// SIMATIC STEP 7 (V5.x) project N2021Andres
// CPU: CPU 314C-2 DP
// station: Hardware
// station: SIMATIC 300 maestro
// station: P_ADR_BUS
// station: P_ADR_BUS
// station: Configuración
// program: Programa S7(1)

SYMBOL_TABLE
"Con_flujo"	C 12	COUNTER
"TempAguaFria"	C 13	COUNTER
"TempAguaCAliente"	C 14	COUNTER
"TempVapor"	C 15	COUNTER
"TempCondensados"	C 16	COUNTER
"EntradasING"	DB 1	DB 1
"Datos1Hp"	DB 3	DB 3	// Datos leidos y enviados al variador de 1 Hp
"Datos2HP"	DB 4	DB 4	// Datos leidos y enviados al variador de 2 Hp
"DatosVarpH"	DB 6	DB 6	// Datos leidos y enviados al variador de 1 Hp
"DatosVarReactor"	DB 7	DB 7	// Datos leidos y enviados al variador de 1 Hp
"CONT_C"	FB 41	FB 41	// Continuous Control
"Escalizaciones"	FC 1	FC 1
"Alarmas"	FC 2	FC 2
"var1hp"	FC 3	FC 3
"var2hp"	FC 4	FC 4
"VarReactor"	FC 5	FC 5
"VarpH"	FC 6	FC 6
"DP_SEND"	FC 15	FC 15	// DP-SEND-Function for  SIMATIC NET CPs
"FT_In"	I 0.0	BOOL
"nivelAltoAlim"	I 2.0	BOOL
"nivelbajoAlim"	I 2.1	BOOL
"termico1hp"	I 2.3	BOOL
"termico2hp"	I 2.4	BOOL
"H_Emergencia"	I 2.5	BOOL
"start1hp"	M 1.0	BOOL
"stop1hp"	M 1.1	BOOL
"recFall1hp"	M 1.2	BOOL
"start2hp"	M 1.3	BOOL
"stop2hp"	M 1.4	BOOL
"recFalla2hp"	M 1.5	BOOL
"ResetSPNivel"	M 1.6	BOOL
"siempreOff"	M 2.0	BOOL
"siempreon"	M 2.1	BOOL
"Cascada"	M 2.2	BOOL
"manpid1"	M 2.3	BOOL
"manpid2"	M 2.4	BOOL
"manpid3"	M 2.5	BOOL
"M_ALLTKpeq"	M 3.0	BOOL
"M_AHLTKpeq"	M 3.1	BOOL
"M_Termico1HP"	M 3.2	BOOL
"M_LT_alto"	M 3.3	BOOL
"M_Termico2HP"	M 3.4	BOOL
"M_H.Emerg"	M 3.5	BOOL
"M_AlarmaSobrepresiòn"	M 3.6	BOOL
"AlamaBitporpresion"	M 3.7	BOOL
"resetTotalFlujo"	M 5.0	BOOL
"startReactor"	M 184.0	BOOL
"StopReactor"	M 184.1	BOOL
"RecFallaReactor"	M 184.2	BOOL
"StartpH"	M 184.3	BOOL
"StoppH"	M 184.4	BOOL
"RecFallapH"	M 184.5	BOOL
"FT_Aire_mA"	MD 132	REAL	// señal escalizada en mA del FT de aire a la salida del tanque
"FlujoAireOutLPM"	MD 136	REAL	// flujo de aire medido con el sensor portatil a la salida de la valvula prop
"VoltReactor"	MD 140	REAL
"CorrReactor"	MD 144	REAL
"FreReactor"	MD 148	REAL
"VoltpH"	MD 152	REAL
"CorrpH"	MD 156	REAL
"FrepH"	MD 160	REAL
"Tiempo"	MD 164	REAL
"Total_litros"	MD 172	REAL
"ohmiosPT100"	MD 176	REAL	// ohmios equivalntes para la temperatura db1.dbd40
"flujo_In_lpm"	MD 180	REAL
"Flujo_Out_lpm"	MD 184	REAL
"fre2hp"	MD 188	REAL
"vol2hp"	MD 192	REAL
"corr2hp"	MD 196	DWORD
"fre1hp"	MD 200	DWORD
"vol1hp"	MD 204	REAL
"corr1hp"	MD 208	DWORD
"LTmA"	MD 212	REAL
"FTmA"	MD 216	REAL
"mA_A_IP"	MD 220	REAL
"mA_A_Valve_Prop"	MD 224	REAL
"FrecuenciaDint2"	MD 228	DINT
"pTmA"	MD 232	REAL
"PT_Out_mA"	MD 236	REAL
"LTpsig"	MD 240	REAL
"PulsosTotal"	MD 244	REAL
"PulsosRata"	MD 248	REAL
"FrecuenciaDint"	MD 252	DINT
"FrecuenciaReal"	MD 256	REAL
"erroresfc"	MW 64	WORD
"fre2hpref"	MW 98	WORD
"fre1hpref"	MW 100	WORD
"freReactorref"	MW 102	WORD
"frepHref"	MW 104	WORD
"CYC_INT2"	OB 32	OB 32	// Cyclic Interrupt 2
"CYC_INT3"	OB 33	OB 33	// Cyclic Interrupt 3
"CYC_INT6"	OB 36	OB 36	// Cyclic Interrupt 6
"CYC_INT8"	OB 38	OB 38	// Cyclic Interrupt 8
"LTint"	PIW 50	INT	// FT ultrasonido de nivel rango 0-60cms
"PTint"	PIW 52	INT	// PT en el tanque rango  0-600mBar
"FTint"	PIW 54	INT	// FT en tuberia rango 0-60LPM
"FT_Aire"	PIW 56	INT	// FT flujo aire portatil 0-20 SLPM
"libre1"	PIW 58	WORD
"IP"	PQW 50	WORD
"PropValve"	PQW 52	WORD
"BalisaLuminosa"	Q 0.3	BOOL
"FREQUENC"	SFB 48	SFB 48	// Frequency measurement module
"WR_REC"	SFC 58	SFC 58	// Write Data Record
"com"	VAT 1	
END_SYMBOL_TABLE

// FB 41: know-how protected block, not included

FUNCTION "Escalizaciones" : VOID	// FC 1
VERSION : 0.1
VAR_TEMP
  TEMP0 : DINT ;
  TEMP1 : REAL ;
  temp2 : DINT ;
END_VAR
BEGIN
NETWORK
TITLE = Escalizamos el transmisor de nivel en cms y en mA
      A     "siempreOff";
      =     L 12.0;
      BLD   103;
      A(;
      A     "siempreOff";
      =     L 12.1;
      BLD   103;
      CALL  FC 105 (
           $1                       := P#P 50.0,
           $2                       := L#1114898432,
           $3                       := L#0,
           $4                       := L 12.1,
           $5                       := "erroresfc",
           $6                       := DB10.DBD 10);
      A     BR;
      );
      JNB   _001;
      CALL  FC 105 (
           $1                       := P#P 50.0,
           $2                       := L#1101004800,
           $3                       := L#1082130432,
           $4                       := L 12.0,
           $5                       := "erroresfc",
           $6                       := "LTmA");
_001: NOP   0;
NETWORK
TITLE = Escalizamos el transmisor de presiòn en mbar, en psig y en mA
      A     "siempreOff";
      =     L 12.0;
      BLD   103;
      A(;
      A     "siempreOff";
      =     L 12.1;
      BLD   103;
      CALL  FC 105 (
           $1                       := P#P 52.0,
           $2                       := L#1142292480,
           $3                       := L#0,
           $4                       := L 12.1,
           $5                       := "erroresfc",
           $6                       := DB9.DBD 10);
      A     BR;
      );
      JNB   _002;
      CALL  FC 105 (
           $1                       := P#P 52.0,
           $2                       := L#1101004800,
           $3                       := L#1082130432,
           $4                       := L 12.0,
           $5                       := "erroresfc",
           $6                       := "pTmA");
_002: NOP   0;
NETWORK
TITLE = Escalizamos el transmisor de flujo ultrasonido en lpm y mA
      A     "siempreOff";
      =     L 12.0;
      BLD   103;
      A(;
      A     "siempreOff";
      =     L 12.1;
      BLD   103;
      CALL  FC 105 (
           $1                       := P#P 54.0,
           $2                       := L#1101004800,
           $3                       := L#1082130432,
           $4                       := L 12.1,
           $5                       := "erroresfc",
           $6                       := "FTmA");
      A     BR;
      );
      JNB   _003;
      CALL  FC 105 (
           $1                       := P#P 54.0,
           $2                       := L#1114636288,
           $3                       := L#0,
           $4                       := L 12.0,
           $5                       := "erroresfc",
           $6                       := DB11.DBD 10);
_003: NOP   0;
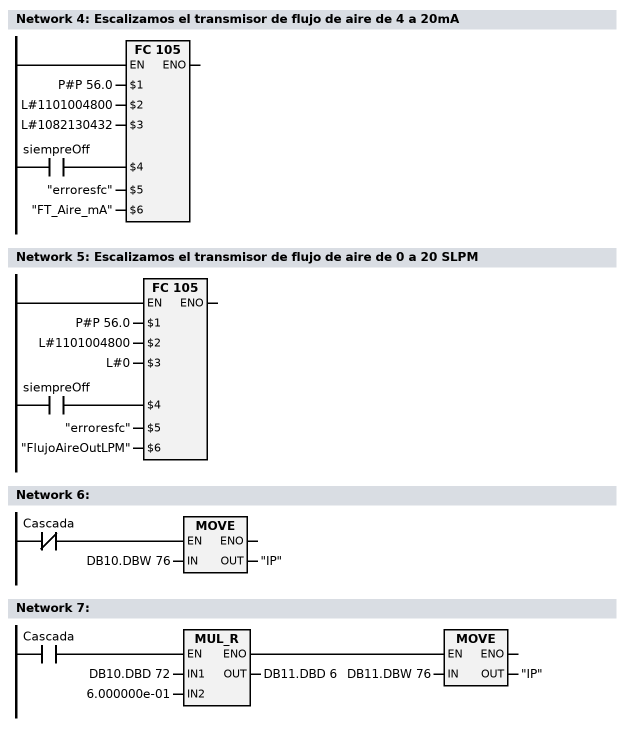
NETWORK
TITLE = Escalizamos el transmisor de flujo de aire de 4 a 20mA
      A     "siempreOff";
      =     L 12.0;
      BLD   103;
      CALL  FC 105 (
           $1                       := P#P 56.0,
           $2                       := L#1101004800,
           $3                       := L#1082130432,
           $4                       := L 12.0,
           $5                       := "erroresfc",
           $6                       := "FT_Aire_mA");
      NOP   0;
NETWORK
TITLE = Escalizamos el transmisor de flujo de aire de 0 a 20 SLPM
      A     "siempreOff";
      =     L 12.0;
      BLD   103;
      CALL  FC 105 (
           $1                       := P#P 56.0,
           $2                       := L#1101004800,
           $3                       := L#0,
           $4                       := L 12.0,
           $5                       := "erroresfc",
           $6                       := "FlujoAireOutLPM");
      NOP   0;
NETWORK
TITLE =
//Si es control de nivel llevamos la salida al IP1
      AN    "Cascada";
      JNB   _004;
      L     DB10.DBW 76;
      T     "IP";
_004: NOP   0;
NETWORK
TITLE =
//LLevamos la salida del control de nivel como setPoint al control de flujo y la 
//salida del control de flujo a la salida fisica
//
      A(;
      A     "Cascada";
      JNB   _005;
      L     DB10.DBD 72;
      L     6.000000e-01;
      *R;
      T     DB11.DBD 6;
      AN    OV;
      SAVE;
      CLR;
_005: A     BR;
      );
      JNB   _006;
      L     DB11.DBW 76;
      T     "IP";
_006: NOP   0;
END_FUNCTION

FUNCTION "Alarmas" : VOID	// FC 2
VERSION : 0.1
BEGIN
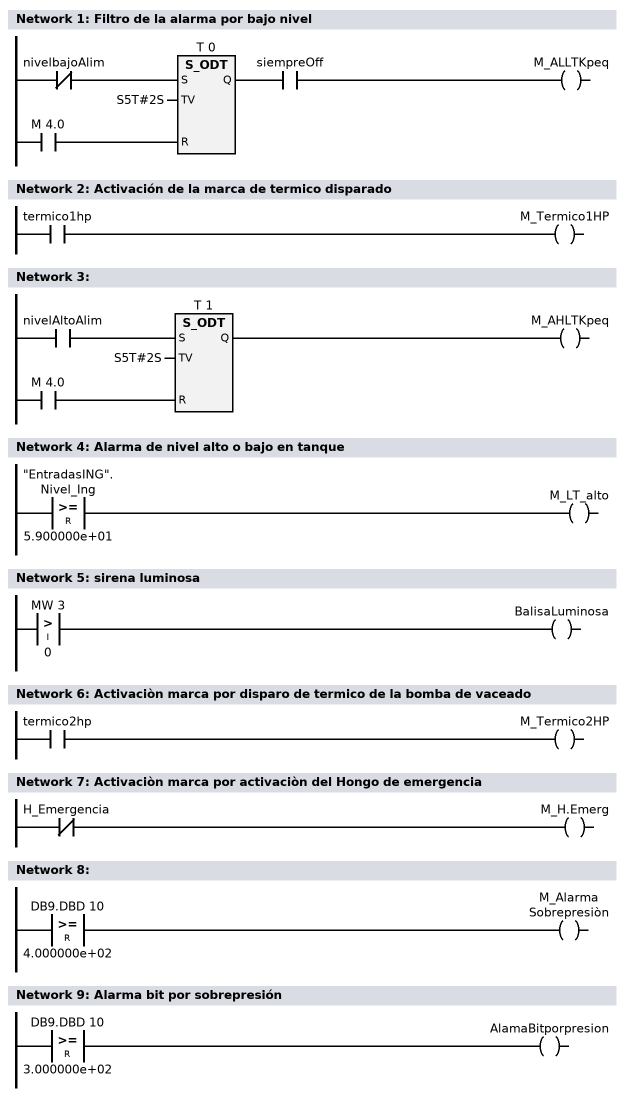
NETWORK
TITLE = Filtro de la alarma por bajo nivel
      A(;
      AN    "nivelbajoAlim";
      L     S5T#2S;
      SD    T 0;
      A     M 4.0;
      R     T 0;
      NOP   0;
      NOP   0;
      A     T 0;
      );
      A     "siempreOff";
      =     "M_ALLTKpeq";
NETWORK
TITLE = Activación de la marca de termico disparado
      A     "termico1hp";
      =     "M_Termico1HP";
NETWORK
TITLE =
//Filtro de la alarma por alto nivel
      A     "nivelAltoAlim";
      L     S5T#2S;
      SD    T 1;
      A     M 4.0;
      R     T 1;
      NOP   0;
      NOP   0;
      A     T 1;
      =     "M_AHLTKpeq";
NETWORK
TITLE = Alarma de nivel alto o bajo en tanque
      L     "EntradasING".Nivel_Ing;
      L     5.900000e+01;
      >=R;
      =     "M_LT_alto";
NETWORK
TITLE = sirena luminosa
      L     MW 3;
      L     0;
      >I;
      =     "BalisaLuminosa";
NETWORK
TITLE = Activaciòn marca por disparo de termico de la bomba de vaceado
      A     "termico2hp";
      =     "M_Termico2HP";
NETWORK
TITLE = Activaciòn marca por activaciòn del Hongo de emergencia
      AN    "H_Emergencia";
      =     "M_H.Emerg";
NETWORK
TITLE =
      L     DB9.DBD 10;
      L     4.000000e+02;
      >=R;
      =     "M_AlarmaSobrepresiòn";
NETWORK
TITLE = Alarma bit por sobrepresión
      L     DB9.DBD 10;
      L     3.000000e+02;
      >=R;
      =     "AlamaBitporpresion";
END_FUNCTION

FUNCTION "var1hp" : VOID	// FC 3
TITLE = Lectura y escritura de datos en el variador de 1Hp
VERSION : 0.1
VAR_TEMP
  temp1_1 : INT ;
  freRef : INT ;
  temp1 : DINT ;
  temp0 : REAL ;
  TempConverDoble : DWORD ;
END_VAR
BEGIN
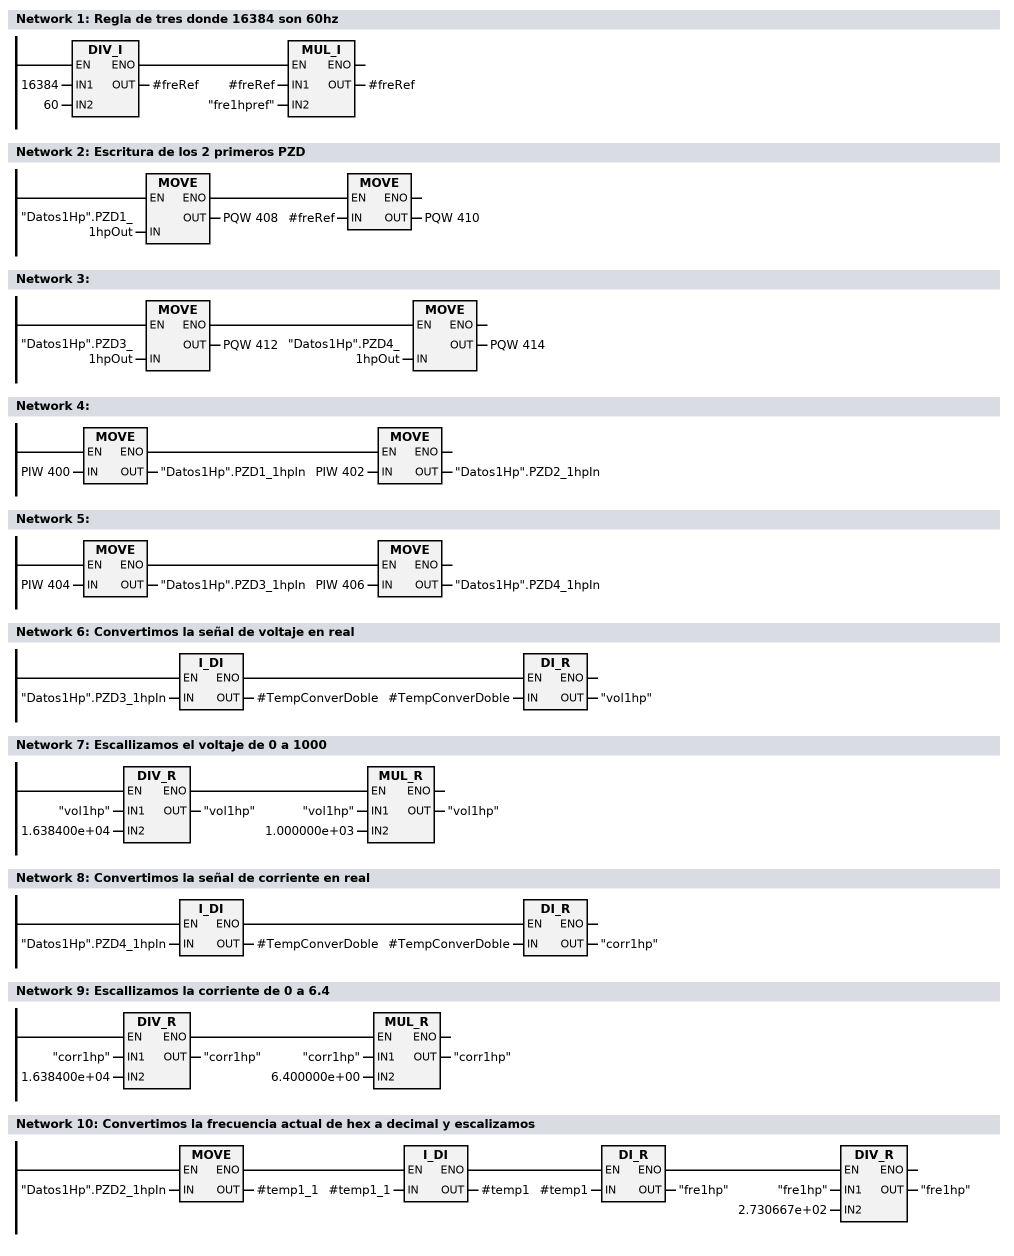
NETWORK
TITLE = Regla de tres donde 16384 son 60hz
      A(;
      L     16384;
      L     60;
      /I;
      T     #freRef;
      AN    OV;
      SAVE;
      CLR;
      A     BR;
      );
      JNB   _001;
      L     #freRef;
      L     "fre1hpref";
      *I;
      T     #freRef;
_001: NOP   0;
NETWORK
TITLE = Escritura de los 2 primeros PZD
//Peticion Dato Alimentacion
      A(;
      L     "Datos1Hp".PZD1_1hpOut;
      T     PQW 408;
      SET;
      SAVE;
      CLR;
      A     BR;
      );
      JNB   _002;
      L     #freRef;
      T     PQW 410;
_002: NOP   0;
NETWORK
TITLE =
//Escritura de los 2 ultimos PZD
      A(;
      L     "Datos1Hp".PZD3_1hpOut;
      T     PQW 412;
      SET;
      SAVE;
      CLR;
      A     BR;
      );
      JNB   _003;
      L     "Datos1Hp".PZD4_1hpOut;
      T     PQW 414;
_003: NOP   0;
NETWORK
TITLE =
//Lectura de los 2 primeros PZD
//
      A(;
      L     PIW 400;
      T     "Datos1Hp".PZD1_1hpIn;
      SET;
      SAVE;
      CLR;
      A     BR;
      );
      JNB   _00b;
      L     PIW 402;
      T     "Datos1Hp".PZD2_1hpIn;
_00b: NOP   0;
NETWORK
TITLE =
//Lectura de los 2 ultimos PZD voltaje y corriente
//
      A(;
      L     PIW 404;
      T     "Datos1Hp".PZD3_1hpIn;
      SET;
      SAVE;
      CLR;
      A     BR;
      );
      JNB   _00d;
      L     PIW 406;
      T     "Datos1Hp".PZD4_1hpIn;
_00d: NOP   0;
NETWORK
TITLE = Convertimos la señal de voltaje en real
      A(;
      L     "Datos1Hp".PZD3_1hpIn;
      ITD;
      T     #TempConverDoble;
      SET;
      SAVE;
      CLR;
      A     BR;
      );
      JNB   _014;
      L     #TempConverDoble;
      DTR;
      T     "vol1hp";
_014: NOP   0;
NETWORK
TITLE = Escallizamos el voltaje de 0 a 1000
      A(;
      L     "vol1hp";
      L     1.638400e+04;
      /R;
      T     "vol1hp";
      AN    OV;
      SAVE;
      CLR;
      A     BR;
      );
      JNB   _015;
      L     "vol1hp";
      L     1.000000e+03;
      *R;
      T     "vol1hp";
_015: NOP   0;
NETWORK
TITLE = Convertimos la señal de corriente en real
      A(;
      L     "Datos1Hp".PZD4_1hpIn;
      ITD;
      T     #TempConverDoble;
      SET;
      SAVE;
      CLR;
      A     BR;
      );
      JNB   _013;
      L     #TempConverDoble;
      DTR;
      T     "corr1hp";
_013: NOP   0;
NETWORK
TITLE = Escallizamos la corriente de 0 a 6.4
      A(;
      L     "corr1hp";
      L     1.638400e+04;
      /R;
      T     "corr1hp";
      AN    OV;
      SAVE;
      CLR;
      A     BR;
      );
      JNB   _007;
      L     "corr1hp";
      L     6.400000e+00;
      *R;
      T     "corr1hp";
_007: NOP   0;
NETWORK
TITLE = Convertimos la frecuencia actual de hex a decimal y escalizamos 
      A(;
      A(;
      A(;
      L     "Datos1Hp".PZD2_1hpIn;
      T     #temp1_1;
      SET;
      SAVE;
      CLR;
      A     BR;
      );
      JNB   _008;
      L     #temp1_1;
      ITD;
      T     #temp1;
      SET;
      SAVE;
      CLR;
_008: A     BR;
      );
      JNB   _009;
      L     #temp1;
      DTR;
      T     "fre1hp";
      SET;
      SAVE;
      CLR;
_009: A     BR;
      );
      JNB   _00a;
      L     "fre1hp";
      L     2.730667e+02;
      /R;
      T     "fre1hp";
_00a: NOP   0;
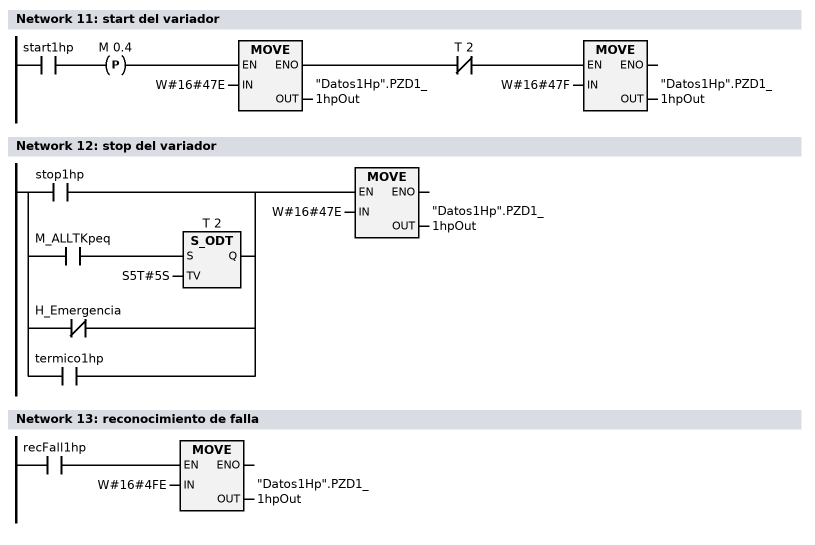
NETWORK
TITLE = start del variador
      A(;
      A     "start1hp";
      FP    M 0.4;
      JNB   _016;
      L     W#16#47E;
      T     "Datos1Hp".PZD1_1hpOut;
      SET;
      SAVE;
      CLR;
_016: A     BR;
      );
      AN    T 2;
      JNB   _017;
      L     W#16#47F;
      T     "Datos1Hp".PZD1_1hpOut;
_017: NOP   0;
NETWORK
TITLE = stop del variador
//paramos la bomba de llenado si el usuario le da la orden o si el nivel cae por 
//5 
//seg en el tanque de alimentaciòn
      A(;
      O     "stop1hp";
      O(;
      A     "M_ALLTKpeq";
      L     S5T#5S;
      SD    T 2;
      NOP   0;
      NOP   0;
      NOP   0;
      A     T 2;
      );
      ON    "H_Emergencia";
      O     "termico1hp";
      );
      JNB   _01b;
      L     W#16#47E;
      T     "Datos1Hp".PZD1_1hpOut;
_01b: NOP   0;
NETWORK
TITLE = reconocimiento de falla
      A     "recFall1hp";
      JNB   _021;
      L     W#16#4FE;
      T     "Datos1Hp".PZD1_1hpOut;
_021: NOP   0;
END_FUNCTION

FUNCTION "var2hp" : VOID	// FC 4
TITLE = Lectura y escritura de datos en el variador de 1Hp
VERSION : 0.1
VAR_TEMP
  temp1_1 : INT ;
  freRef : INT ;
  temp1 : DINT ;
  temp0 : REAL ;
  TempConverDoble : DWORD ;
END_VAR
BEGIN
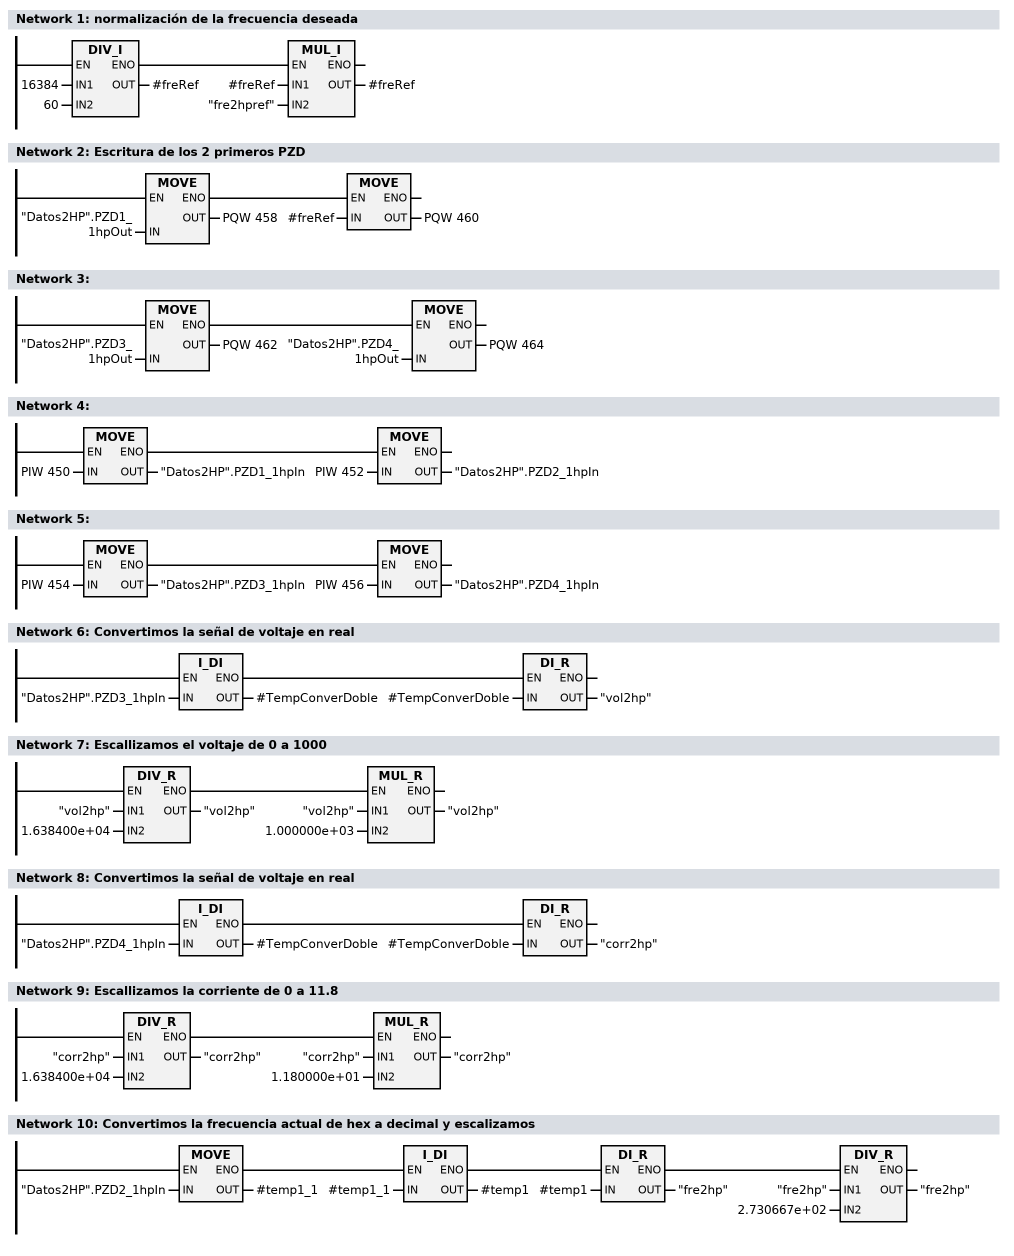
NETWORK
TITLE = normalización de la frecuencia deseada 
      A(;
      L     16384;
      L     60;
      /I;
      T     #freRef;
      AN    OV;
      SAVE;
      CLR;
      A     BR;
      );
      JNB   _003;
      L     #freRef;
      L     "fre2hpref";
      *I;
      T     #freRef;
_003: NOP   0;
NETWORK
TITLE = Escritura de los 2 primeros PZD
//Peticion Dato Alimentacion
      A(;
      L     "Datos2HP".PZD1_1hpOut;
      T     PQW 458;
      SET;
      SAVE;
      CLR;
      A     BR;
      );
      JNB   _001;
      L     #freRef;
      T     PQW 460;
_001: NOP   0;
NETWORK
TITLE =
//Escritura de los 2 ultimos PZD
      A(;
      L     "Datos2HP".PZD3_1hpOut;
      T     PQW 462;
      SET;
      SAVE;
      CLR;
      A     BR;
      );
      JNB   _005;
      L     "Datos2HP".PZD4_1hpOut;
      T     PQW 464;
_005: NOP   0;
NETWORK
TITLE =
//Lectura de los 2 primeros PZD
//
      A(;
      L     PIW 450;
      T     "Datos2HP".PZD1_1hpIn;
      SET;
      SAVE;
      CLR;
      A     BR;
      );
      JNB   _006;
      L     PIW 452;
      T     "Datos2HP".PZD2_1hpIn;
_006: NOP   0;
NETWORK
TITLE =
//Lectura de los 2 ultimos PZD voltaje y corriente
//
      A(;
      L     PIW 454;
      T     "Datos2HP".PZD3_1hpIn;
      SET;
      SAVE;
      CLR;
      A     BR;
      );
      JNB   _007;
      L     PIW 456;
      T     "Datos2HP".PZD4_1hpIn;
_007: NOP   0;
NETWORK
TITLE = Convertimos la señal de voltaje en real
      A(;
      L     "Datos2HP".PZD3_1hpIn;
      ITD;
      T     #TempConverDoble;
      SET;
      SAVE;
      CLR;
      A     BR;
      );
      JNB   _014;
      L     #TempConverDoble;
      DTR;
      T     "vol2hp";
_014: NOP   0;
NETWORK
TITLE = Escallizamos el voltaje de 0 a 1000
      A(;
      L     "vol2hp";
      L     1.638400e+04;
      /R;
      T     "vol2hp";
      AN    OV;
      SAVE;
      CLR;
      A     BR;
      );
      JNB   _00b;
      L     "vol2hp";
      L     1.000000e+03;
      *R;
      T     "vol2hp";
_00b: NOP   0;
NETWORK
TITLE = Convertimos la señal de voltaje en real
      A(;
      L     "Datos2HP".PZD4_1hpIn;
      ITD;
      T     #TempConverDoble;
      SET;
      SAVE;
      CLR;
      A     BR;
      );
      JNB   _013;
      L     #TempConverDoble;
      DTR;
      T     "corr2hp";
_013: NOP   0;
NETWORK
TITLE = Escallizamos la corriente de 0 a 11.8
      A(;
      L     "corr2hp";
      L     1.638400e+04;
      /R;
      T     "corr2hp";
      AN    OV;
      SAVE;
      CLR;
      A     BR;
      );
      JNB   _022;
      L     "corr2hp";
      L     1.180000e+01;
      *R;
      T     "corr2hp";
_022: NOP   0;
NETWORK
TITLE = Convertimos la frecuencia actual de hex a decimal y escalizamos 
      A(;
      A(;
      A(;
      L     "Datos2HP".PZD2_1hpIn;
      T     #temp1_1;
      SET;
      SAVE;
      CLR;
      A     BR;
      );
      JNB   _017;
      L     #temp1_1;
      ITD;
      T     #temp1;
      SET;
      SAVE;
      CLR;
_017: A     BR;
      );
      JNB   _01b;
      L     #temp1;
      DTR;
      T     "fre2hp";
      SET;
      SAVE;
      CLR;
_01b: A     BR;
      );
      JNB   _01d;
      L     "fre2hp";
      L     2.730667e+02;
      /R;
      T     "fre2hp";
_01d: NOP   0;
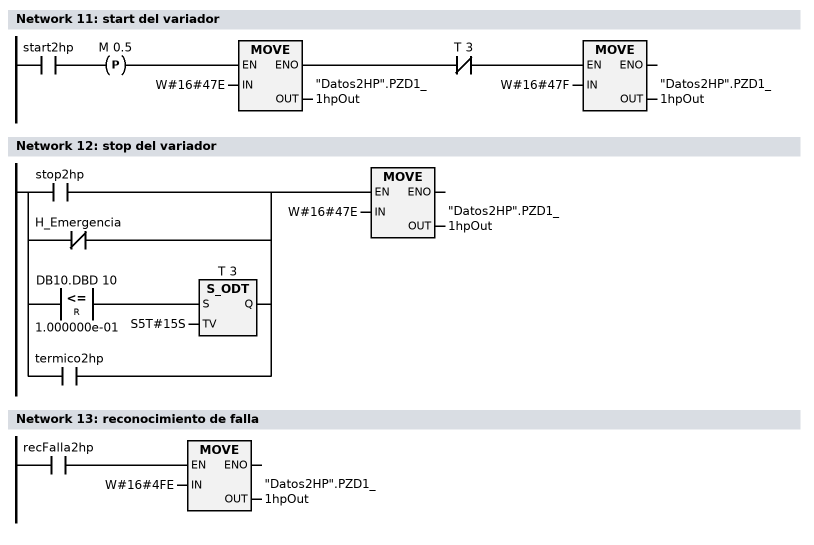
NETWORK
TITLE = start del variador
      A(;
      A     "start2hp";
      FP    M 0.5;
      JNB   _01e;
      L     W#16#47E;
      T     "Datos2HP".PZD1_1hpOut;
      SET;
      SAVE;
      CLR;
_01e: A     BR;
      );
      AN    T 3;
      JNB   _01f;
      L     W#16#47F;
      T     "Datos2HP".PZD1_1hpOut;
_01f: NOP   0;
NETWORK
TITLE = stop del variador
      A(;
      O     "stop2hp";
      ON    "H_Emergencia";
      O(;
      A(;
      L     DB10.DBD 10;
      L     1.000000e-01;
      <=R;
      );
      L     S5T#15S;
      SD    T 3;
      NOP   0;
      NOP   0;
      NOP   0;
      A     T 3;
      );
      O     "termico2hp";
      );
      JNB   _021;
      L     W#16#47E;
      T     "Datos2HP".PZD1_1hpOut;
_021: NOP   0;
NETWORK
TITLE = reconocimiento de falla
      A     "recFalla2hp";
      JNB   _023;
      L     W#16#4FE;
      T     "Datos2HP".PZD1_1hpOut;
_023: NOP   0;
END_FUNCTION

// FC 105: know-how protected block, not included

DATA_BLOCK "EntradasING"	// DB 1
VERSION : 0.1
  STRUCT
   LimSupLT : REAL  := 6.100000e+001;
   LimInfLT : REAL ;
   LimSupPT : REAL  := 6.000000e+002;
   LimInfPT : REAL ;
   Nivel_Ing : REAL ;
   Presin_Ing : REAL ;
   STAT6 : REAL  := 2.000000e+001;
   STAT7 : REAL  := 4.000000e+000;
   STAT8 : REAL  := 6.000000e+001;
   STAT9 : REAL ;
   STAT10 : REAL ;
   STAT11 : REAL ;
   STAT12 : REAL ;
   STAT13 : REAL ;
   STAT14 : REAL ;
   STAT15 : REAL ;
   STAT16 : REAL ;
   STAT17 : REAL ;
   STAT18 : REAL ;
   STAT19 : REAL ;
   STAT20 : REAL ;
   STAT21 : REAL ;
   STAT22 : REAL ;
  END_STRUCT ;	
BEGIN
   LimSupLT := 6.100000e+01;
   LimSupPT := 1.000000e+02;
   Nivel_Ing := 5.000000e+01;
   STAT6 := 2.000000e+02;
   STAT9 := 2.680000e+01;
   STAT10 := 4.780000e+01;
   STAT11 := 2.850000e+01;
   STAT12 := 2.780000e+01;
   STAT13 := 3.276700e+03;
   STAT14 := 3.276700e+03;
   STAT15 := 3.276700e+03;
   STAT16 := 3.276700e+03;
END_DATA_BLOCK

DATA_BLOCK "Datos1Hp"	// DB 3
VERSION : 0.1
  STRUCT
   PZD1_1hpIn : WORD ;
   PZD2_1hpIn : WORD ;
   PZD3_1hpIn : WORD ;
   PZD4_1hpIn : WORD ;
   PZD1_1hpOut : WORD ;
   PZD2_1hpOut : WORD ;
   PZD3_1hpOut : WORD ;
   PZD4_1hpOut : WORD ;
   PKW1_1hpIn : WORD ;
   PKW2_1hpIn : WORD ;
   PKW3_1hpIn : WORD ;
   PKW4_1hpIn : WORD ;
   PKW1_1hpOut : WORD ;
   PKW2_1hpOut : WORD ;
   PKW3_1hpOut : WORD ;
   PKW4_1hpOut : WORD ;
  END_STRUCT ;	
BEGIN
   PZD1_1hpIn := W#16#FB31;
   PZD1_1hpOut := W#16#47E;
END_DATA_BLOCK

DATA_BLOCK "Datos2HP"	// DB 4
VERSION : 0.1
  STRUCT
   PZD1_1hpIn : WORD ;
   PZD2_1hpIn : WORD ;
   PZD3_1hpIn : WORD ;
   PZD4_1hpIn : WORD ;
   PZD1_1hpOut : WORD ;
   PZD2_1hpOut : WORD ;
   PZD3_1hpOut : WORD ;
   PZD4_1hpOut : WORD ;
   PKW1_1hpIn : WORD ;
   PKW2_1hpIn : WORD ;
   PKW3_1hpIn : WORD ;
   PKW4_1hpIn : WORD ;
   PKW1_1hpOut : WORD ;
   PKW2_1hpOut : WORD ;
   PKW3_1hpOut : WORD ;
   PKW4_1hpOut : WORD ;
  END_STRUCT ;	
BEGIN
   PZD1_1hpIn := W#16#FB31;
   PZD1_1hpOut := W#16#47E;
END_DATA_BLOCK

DATA_BLOCK DB 8
AUTHOR : SIMATIC
FAMILY : TEC_FUNC
VERSION : 0.0
"FREQUENC"
BEGIN
END_DATA_BLOCK

DATA_BLOCK DB 9
AUTHOR : SIMATIC
FAMILY : ICONT
VERSION : 0.0
"CONT_C"
BEGIN
END_DATA_BLOCK

DATA_BLOCK DB 10
AUTHOR : SIMATIC
FAMILY : ICONT
VERSION : 0.0
"CONT_C"
BEGIN
END_DATA_BLOCK

DATA_BLOCK DB 11
AUTHOR : SIMATIC
FAMILY : ICONT
VERSION : 0.0
"CONT_C"
BEGIN
END_DATA_BLOCK

ORGANIZATION_BLOCK OB 1
TITLE = "Main Program Sweep (Cycle)"
VERSION : 0.1
VAR_TEMP
  TEMP0 : BYTE ;
  TEMP1 : BYTE ;
  TEMP2 : BYTE ;
  TEMP3 : BYTE ;
  TEMP4 : BYTE ;
  TEMP5 : BYTE ;
  TEMP6 : INT ;
  TEMP7 : INT ;
  TEMP8 : INT ;
  TEMP9 : DATE_AND_TIME ;
  TEMP10 : REAL ;
  temp2_1 : DINT ;
  tempReal : REAL ;
END_VAR
BEGIN
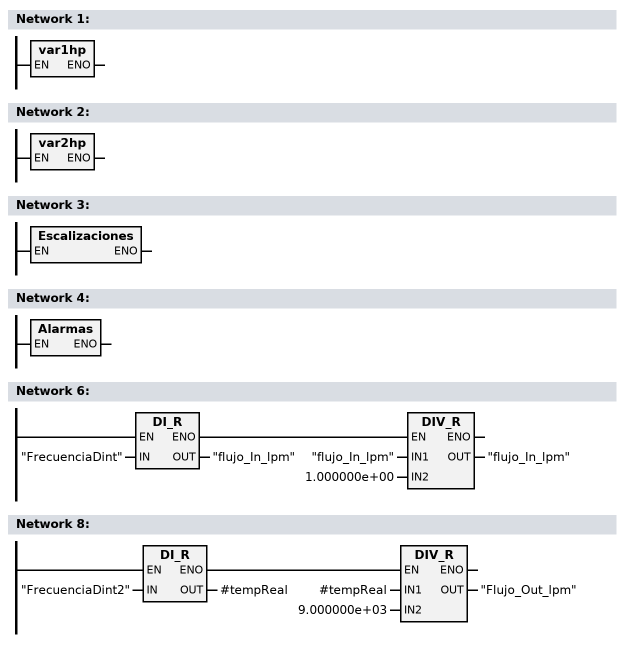
NETWORK
TITLE =
      CALL  "var1hp";
      NOP   0;
NETWORK
TITLE =
      CALL  "var2hp";
      NOP   0;
NETWORK
TITLE =
      CALL  "Escalizaciones";
      NOP   0;
NETWORK
TITLE =
      CALL  "Alarmas";
      NOP   0;
NETWORK
TITLE =
      A     "siempreon";
      =     L 32.0;
      BLD   103;
      BLD   9;
      =     L 37.0;
      CDB;
      OPN   DI 8;
      TAR2  LD 33;
      L     PIW 768;
      T     DIW 0;
      L     1;
      T     DIW 2;
      A     L 32.0;
      =     DIX 4.0;
      LAR2  P#DBX 0.0;
      UC    "FREQUENC";
      LAR2  LD 33;
      L     DID 14;
      T     "FrecuenciaDint";
      CDB;
      BLD   10;
      NOP   0;
NETWORK
TITLE =
      A(;
      L     "FrecuenciaDint";
      DTR;
      T     "flujo_In_lpm";
      SET;
      SAVE;
      CLR;
      A     BR;
      );
      JNB   _001;
      L     "flujo_In_lpm";
      L     1.000000e+00;
      /R;
      T     "flujo_In_lpm";
_001: NOP   0;
NETWORK
TITLE =
      A     "siempreon";
      =     L 32.0;
      BLD   103;
      BLD   9;
      =     L 37.0;
      CDB;
      OPN   DI 8;
      TAR2  LD 33;
      L     PIW 770;
      T     DIW 0;
      L     0;
      T     DIW 2;
      A     L 32.0;
      =     DIX 4.0;
      LAR2  P#DBX 0.0;
      UC    "FREQUENC";
      LAR2  LD 33;
      L     DID 14;
      T     "FrecuenciaDint2";
      CDB;
      BLD   10;
      NOP   0;
NETWORK
TITLE =
      A(;
      L     "FrecuenciaDint2";
      DTR;
      T     #tempReal;
      SET;
      SAVE;
      CLR;
      A     BR;
      );
      JNB   _002;
      L     #tempReal;
      L     9.000000e+03;
      /R;
      T     "Flujo_Out_lpm";
_002: NOP   0;
END_ORGANIZATION_BLOCK

ORGANIZATION_BLOCK OB 35
VERSION : 0.1
VAR_TEMP
  TEMP0 : BYTE ;
  TEMP1 : BYTE ;
  TEMP2 : BYTE ;
  TEMP3 : BYTE ;
  TEMP4 : BYTE ;
  TEMP5 : BYTE ;
  TEMP6 : WORD ;
  TEMP7 : INT ;
  TEMP8 : INT ;
  TEMP9 : DATE_AND_TIME ;
  TEMP10 : REAL ;
  tempcalc : INT ;
  TEMP11 : REAL ;
  Temp12 : REAL ;
END_VAR
BEGIN
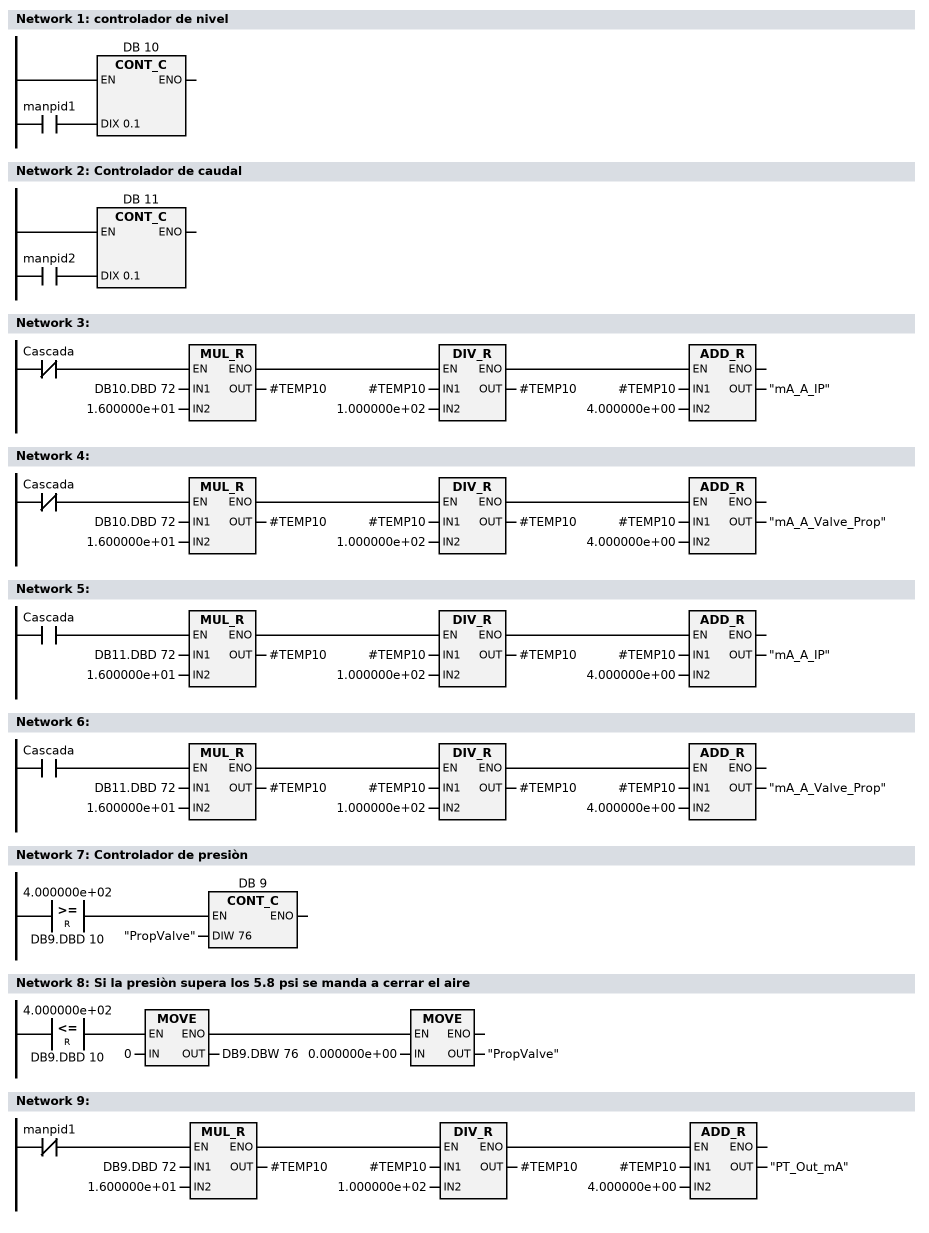
NETWORK
TITLE = controlador de nivel
      A     "manpid1";
      =     L 34.1;
      BLD   103;
      CALL  "CONT_C" , DB 10 (
           DIX 0.1                  := L 34.1);
      NOP   0;
NETWORK
TITLE = Controlador de caudal
      A     "manpid2";
      =     L 34.1;
      BLD   103;
      CALL  "CONT_C" , DB 11 (
           DIX 0.1                  := L 34.1);
      NOP   0;
NETWORK
TITLE =
      A(;
      A(;
      AN    "Cascada";
      JNB   _001;
      L     DB10.DBD 72;
      L     1.600000e+01;
      *R;
      T     #TEMP10;
      AN    OV;
      SAVE;
      CLR;
_001: A     BR;
      );
      JNB   _002;
      L     #TEMP10;
      L     1.000000e+02;
      /R;
      T     #TEMP10;
      AN    OV;
      SAVE;
      CLR;
_002: A     BR;
      );
      JNB   _003;
      L     #TEMP10;
      L     4.000000e+00;
      +R;
      T     "mA_A_IP";
_003: NOP   0;
NETWORK
TITLE =
      A(;
      A(;
      AN    "Cascada";
      JNB   _004;
      L     DB10.DBD 72;
      L     1.600000e+01;
      *R;
      T     #TEMP10;
      AN    OV;
      SAVE;
      CLR;
_004: A     BR;
      );
      JNB   _005;
      L     #TEMP10;
      L     1.000000e+02;
      /R;
      T     #TEMP10;
      AN    OV;
      SAVE;
      CLR;
_005: A     BR;
      );
      JNB   _006;
      L     #TEMP10;
      L     4.000000e+00;
      +R;
      T     "mA_A_Valve_Prop";
_006: NOP   0;
NETWORK
TITLE =
      A(;
      A(;
      A     "Cascada";
      JNB   _007;
      L     DB11.DBD 72;
      L     1.600000e+01;
      *R;
      T     #TEMP10;
      AN    OV;
      SAVE;
      CLR;
_007: A     BR;
      );
      JNB   _008;
      L     #TEMP10;
      L     1.000000e+02;
      /R;
      T     #TEMP10;
      AN    OV;
      SAVE;
      CLR;
_008: A     BR;
      );
      JNB   _009;
      L     #TEMP10;
      L     4.000000e+00;
      +R;
      T     "mA_A_IP";
_009: NOP   0;
NETWORK
TITLE =
      A(;
      A(;
      A     "Cascada";
      JNB   _00a;
      L     DB11.DBD 72;
      L     1.600000e+01;
      *R;
      T     #TEMP10;
      AN    OV;
      SAVE;
      CLR;
_00a: A     BR;
      );
      JNB   _00b;
      L     #TEMP10;
      L     1.000000e+02;
      /R;
      T     #TEMP10;
      AN    OV;
      SAVE;
      CLR;
_00b: A     BR;
      );
      JNB   _00c;
      L     #TEMP10;
      L     4.000000e+00;
      +R;
      T     "mA_A_Valve_Prop";
_00c: NOP   0;
NETWORK
TITLE = Controlador de presiòn
//Si la presión es menor a 400mbar (5.8psig) activamos el PID
      A(;
      L     4.000000e+02;
      L     DB9.DBD 10;
      >=R;
      );
      JNB   _00d;
      CALL  "CONT_C" , DB 9 (
           DIW 76                   := "PropValve");
_00d: NOP   0;
NETWORK
TITLE = Si la presiòn supera los 5.8 psi se manda a cerrar el aire 
      A(;
      A(;
      L     4.000000e+02;
      L     DB9.DBD 10;
      <=R;
      );
      JNB   _00e;
      L     0;
      T     DB9.DBW 76;
      SET;
      SAVE;
      CLR;
_00e: A     BR;
      );
      JNB   _00f;
      L     0.000000e+00;
      T     "PropValve";
_00f: NOP   0;
NETWORK
TITLE =
      A(;
      A(;
      AN    "manpid1";
      JNB   _010;
      L     DB9.DBD 72;
      L     1.600000e+01;
      *R;
      T     #TEMP10;
      AN    OV;
      SAVE;
      CLR;
_010: A     BR;
      );
      JNB   _011;
      L     #TEMP10;
      L     1.000000e+02;
      /R;
      T     #TEMP10;
      AN    OV;
      SAVE;
      CLR;
_011: A     BR;
      );
      JNB   _012;
      L     #TEMP10;
      L     4.000000e+00;
      +R;
      T     "PT_Out_mA";
_012: NOP   0;
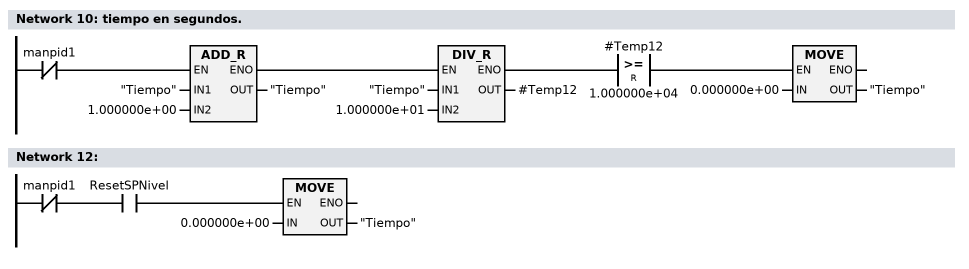
NETWORK
TITLE = tiempo en segundos.
      A(;
      A(;
      AN    "manpid1";
      JNB   _013;
      L     "Tiempo";
      L     1.000000e+00;
      +R;
      T     "Tiempo";
      AN    OV;
      SAVE;
      CLR;
_013: A     BR;
      );
      JNB   _014;
      L     "Tiempo";
      L     1.000000e+01;
      /R;
      T     #Temp12;
      AN    OV;
      SAVE;
      CLR;
_014: A     BR;
      );
      A(;
      L     #Temp12;
      L     1.000000e+04;
      >=R;
      );
      JNB   _015;
      L     0.000000e+00;
      T     "Tiempo";
_015: NOP   0;
NETWORK
TITLE = S.P senoidal de nivel.
// (network holds code this reader does not know; not shown)
NETWORK
TITLE =
      AN    "manpid1";
      A     "ResetSPNivel";
      JNB   _01b;
      L     0.000000e+00;
      T     "Tiempo";
_01b: NOP   0;
END_ORGANIZATION_BLOCK

ORGANIZATION_BLOCK OB 82
VERSION : 0.1
VAR_TEMP
  TEMP0 : BYTE ;
  TEMP1 : BYTE ;
  TEMP2 : BYTE ;
  TEMP3 : BYTE ;
  TEMP4 : BYTE ;
  TEMP5 : BYTE ;
  TEMP6 : WORD ;
  TEMP7 : BOOL ;
  TEMP8 : BOOL ;
  TEMP9 : BOOL ;
  TEMP10 : BOOL ;
  TEMP11 : BOOL ;
  TEMP12 : BOOL ;
  TEMP13 : BOOL ;
  TEMP14 : BOOL ;
  TEMP15 : BYTE ;
  TEMP16 : BOOL ;
  TEMP17 : BOOL ;
  TEMP18 : BOOL ;
  TEMP19 : BOOL ;
  TEMP20 : BOOL ;
  TEMP21 : BOOL ;
  TEMP22 : BOOL ;
  TEMP23 : BOOL ;
  TEMP24 : BOOL ;
  TEMP25 : BOOL ;
  TEMP26 : BOOL ;
  TEMP27 : BOOL ;
  TEMP28 : BOOL ;
  TEMP29 : BOOL ;
  TEMP30 : BOOL ;
  TEMP31 : BOOL ;
  TEMP32 : DATE_AND_TIME ;
END_VAR
BEGIN
// (block stored without names or comments; labels and parameter names are numbered)
END_ORGANIZATION_BLOCK

ORGANIZATION_BLOCK OB 85
VERSION : 0.1
VAR_TEMP
  TEMP0 : BYTE ;
  TEMP1 : BYTE ;
  TEMP2 : BYTE ;
  TEMP3 : BYTE ;
  TEMP4 : BYTE ;
  TEMP5 : BYTE ;
  TEMP6 : INT ;
  TEMP7 : BYTE ;
  TEMP8 : BYTE ;
  TEMP9 : BYTE ;
  TEMP10 : BYTE ;
  TEMP11 : DATE_AND_TIME ;
END_VAR
BEGIN
// (block stored without names or comments; labels and parameter names are numbered)
END_ORGANIZATION_BLOCK

ORGANIZATION_BLOCK OB 86
VERSION : 0.1
VAR_TEMP
  TEMP0 : BYTE ;
  TEMP1 : BYTE ;
  TEMP2 : BYTE ;
  TEMP3 : BYTE ;
  TEMP4 : BYTE ;
  TEMP5 : BYTE ;
  TEMP6 : WORD ;
  TEMP7 : ARRAY  [0 .. 31 ] OF BOOL ;
  TEMP8 : DATE_AND_TIME ;
END_VAR
BEGIN
// (block stored without names or comments; labels and parameter names are numbered)
END_ORGANIZATION_BLOCK

ORGANIZATION_BLOCK OB 100
VERSION : 0.1
VAR_TEMP
  TEMP0 : BYTE ;
  TEMP1 : BYTE ;
  TEMP2 : BYTE ;
  TEMP3 : BYTE ;
  TEMP4 : BYTE ;
  TEMP5 : BYTE ;
  TEMP6 : WORD ;
  TEMP7 : DWORD ;
  TEMP8 : DATE_AND_TIME ;
END_VAR
BEGIN
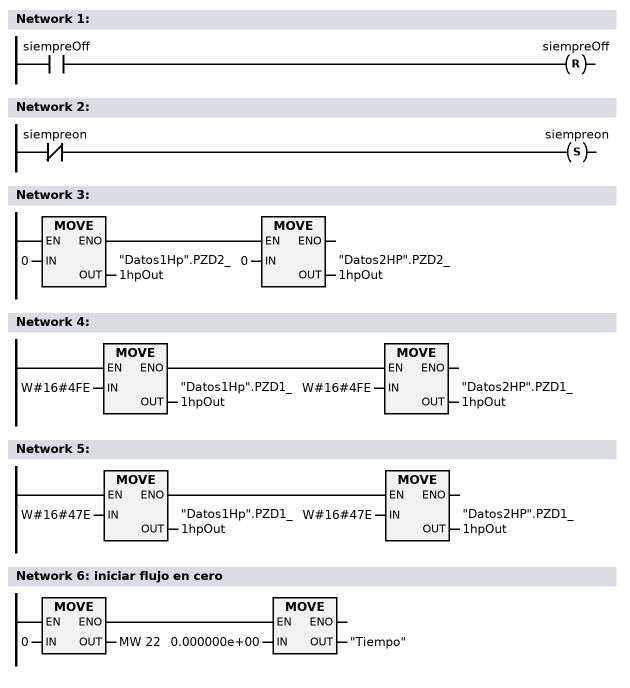
NETWORK
TITLE =
      A     "siempreOff";
      R     "siempreOff";
NETWORK
TITLE =
      AN    "siempreon";
      S     "siempreon";
NETWORK
TITLE =
      A(;
      L     0;
      T     "Datos1Hp".PZD2_1hpOut;
      SET;
      SAVE;
      CLR;
      A     BR;
      );
      JNB   _001;
      L     0;
      T     "Datos2HP".PZD2_1hpOut;
_001: NOP   0;
NETWORK
TITLE =
      A(;
      L     W#16#4FE;
      T     "Datos1Hp".PZD1_1hpOut;
      SET;
      SAVE;
      CLR;
      A     BR;
      );
      JNB   _002;
      L     W#16#4FE;
      T     "Datos2HP".PZD1_1hpOut;
_002: NOP   0;
NETWORK
TITLE =
      A(;
      L     W#16#47E;
      T     "Datos1Hp".PZD1_1hpOut;
      SET;
      SAVE;
      CLR;
      A     BR;
      );
      JNB   _003;
      L     W#16#47E;
      T     "Datos2HP".PZD1_1hpOut;
_003: NOP   0;
NETWORK
TITLE = iniciar flujo en cero
      A(;
      L     0;
      T     MW 22;
      SET;
      SAVE;
      CLR;
      A     BR;
      );
      JNB   _004;
      L     0.000000e+00;
      T     "Tiempo";
_004: NOP   0;
END_ORGANIZATION_BLOCK
